(* IEC 61131-3 sources: POMIRTS_lab3/AS/Library_2/MTRegister/V2.00.0, 3 files *)

(* ---- MTRegister.typ ---- *)
TYPE
	MTRegisterControllerInternalType : 	STRUCT  (*Data for internal use.*)
		CycleTime : REAL; (*Task cycle time. Unit: [s].*)
		ImageLength : REAL; (*Data for internal use.*)
		WebLength : REAL; (*Data for internal use.*)
		SensorPosition : REAL; (*Data for internal use.*)
		MaxVelocityCorrection : REAL; (*Data for internal use.*)
		ResponseRate : REAL; (*Data for internal use.*)
		ResponseOvershoot : REAL; (*Data for internal use.*)
		PrefilterOut : REAL; (*Data for internal use.*)
		ControlStateVariable : REAL; (*Data for internal use.*)
		ControllerParameter : ARRAY[0..2]OF REAL; (*Data for internal use.*)
		ActSystemSampleTime : REAL; (*Data for internal use.*)
		UpdateParametersValid : BOOL; (*Data for internal use.*)
		InitParametersValid : BOOL; (*Data for internal use.*)
		ParametersValid : BOOL; (*Data for internal use.*)
		EnableOld : BOOL; (*Data for internal use.*)
		UpdateOld : BOOL; (*Data for internal use.*)
		InitControllerOld : BOOL; (*Data for internal use.*)
		TriggerOld : BOOL; (*Data for internal use.*)
		ResetOld : BOOL; (*Data for internal use.*)
	END_STRUCT;
	MTRegisterControlModeEnum :
		( (*Mode for the longitudinal register error.*)
		mtPRN_KEY_COLOR := 0, (*Key color mode.*)
		mtPRN_SEQUENTIAL_COLOR := 1 (*Sequential color mode.*)
		);
	MTRegisterDecouplingInternalType : 	STRUCT  (*Data for internal use.*)
		CycleTime : REAL; (*Task cycle time. Unit: [s].*)
		ParametersValid : BOOL; (*Data for internal use.*)
		UpdateOld : BOOL; (*Data for internal use.*)
		EnableOld : {REDUND_UNREPLICABLE} BOOL; (*Data for internal use.*)
		Parameters : {REDUND_UNREPLICABLE} MTRegisterSystemType; (*Data for internal use.*)
		Strain : ARRAY[0..19]OF REAL; (*Data for internal use.*)
		DelayedStrain : ARRAY[0..19]OF REAL; (*Data for internal use.*)
		DelayedChangingStrain : ARRAY[0..19]OF REAL; (*Data for internal use.*)
		NumberOfBufferElements : UINT; (*Data for internal use.*)
		UpdateEpsBuffer : ARRAY[0..18]OF BOOL; (*Data for internal use.*)
		UpdateEpsDerBuffer : ARRAY[0..18]OF BOOL; (*Data for internal use.*)
		EpsBuffer : ARRAY[0..18]OF MTRegisterTransDelayBufferType; (*Data for internal use.*)
		EpsDerBuffer : ARRAY[0..18]OF MTRegisterTransDelayBufferType; (*Data for internal use.*)
		TransportDelayDerivation : ARRAY[0..18]OF REAL; (*Data for internal use.*)
	END_STRUCT;
	MTRegisterSimulationModelIntType : 	STRUCT  (*Data for internal use.*)
		CycleTime : REAL; (*Task cycle time. Unit: [s].*)
		ParametersValid : BOOL; (*Data for internal use.*)
		UpdateOld : BOOL; (*Data for internal use.*)
		EnableOld : {REDUND_UNREPLICABLE} BOOL; (*Data for internal use.*)
		Parameters : {REDUND_UNREPLICABLE} MTRegisterSimulationModelType; (*Data for internal use.*)
		Strain : ARRAY[0..19]OF LREAL; (*Data for internal use.*)
		DelayedStrain : ARRAY[0..19]OF LREAL; (*Data for internal use.*)
		KeyError : ARRAY[0..19]OF REAL; (*Data for internal use.*)
		SequentialError : ARRAY[0..19]OF REAL; (*Data for internal use.*)
		MaterialBreak : ARRAY[0..19]OF BOOL; (*Data for internal use.*)
		RestOfMaterial : ARRAY[0..19]OF REAL; (*Data for internal use.*)
		RegisterError : ARRAY[0..19]OF REAL; (*Data for internal use.*)
		DeltaPos : ARRAY[0..19]OF REAL; (*Data for internal use.*)
		Trigger : ARRAY[0..19]OF BOOL; (*Data for internal use.*)
		NumberEpsBufferElements : USINT; (*Data for internal use.*)
		UpdateEpsBuffer : ARRAY[0..18]OF BOOL; (*Data for internal use.*)
		EpsBuffer : ARRAY[0..18]OF MTRegisterTransDelayLRBufferType; (*Data for internal use.*)
	END_STRUCT;
	MTRegisterSimulationModelType : 	STRUCT  (*Parameter for the simulation model.*)
		NumberOfPrintingUnits : USINT; (*Number of printing units.*)
		ImageLength : DINT; (*Circumference of printing cylinders.*)
		WebLength : ARRAY[0..19]OF DINT; (*Web length between PU#i and PU#i-1. Unit: [µm].*)
		SensorPosition : ARRAY[0..19]OF DINT; (*Distance from printing unit to register mark sensor LSi. Unit: [µm].*)
		Mode : ARRAY[0..19]OF MTRegisterControlModeEnum; (*Control mode array.*)
		TensionIn : REAL; (*Feed tension prior to the first printing unit. Unit: [N].*)
		Noise : BOOL; (*Measurement noise is enabled or disabled.*)
	END_STRUCT;
	MTRegisterSystemType : 	STRUCT  (*System parameters for the decoupling.*)
		NumberOfPrintingUnits : USINT; (*Number of printing units. *)
		WebLength : ARRAY[0..19]OF DINT; (*Web length between PU#i und PU#i-1. Unit: [µm].*)
		Mode : ARRAY[0..19]OF MTRegisterControlModeEnum; (*Control mode array.*)
		AccelerationCompensation : BOOL; (*Compensation of additional acceleration terms.*)
	END_STRUCT;
	MTRegisterTransDelayBufferType : 	STRUCT  (*Buffer parameters for the transport delay.*)
		NumberOfBufferElements : UDINT; (*Data for internal use.*)
		CurrentIndex : UDINT; (*Data for internal use.*)
		DelayIndex : UDINT; (*Data for internal use.*)
		DiffIndex : DINT; (*Data for internal use.*)
		Integration : LREAL; (*Data for internal use.*)
		DataIn : REFERENCE TO REAL; (*Data for internal use.*)
		DataTt : REFERENCE TO REAL; (*Data for internal use.*)
		TimeDelay : REAL; (*Data for internal use.*)
		TransportDelay : REAL; (*Data for internal use.*)
		TransportDelayDerivation : REAL; (*Data for internal use.*)
		MaxDelayTime : REAL; (*Data for internal use.*)
	END_STRUCT;
	MTRegisterTransDelayLRBufferType : 	STRUCT  (*Buffer parameters for the transport delay.*)
		NumberOfBufferElements : UDINT; (*Data for internal use.*)
		CurrentIndex : UDINT; (*Data for internal use.*)
		DelayIndex : UDINT; (*Data for internal use.*)
		DiffIndex : DINT; (*Data for internal use.*)
		Integration : LREAL; (*Data for internal use.*)
		DataIn : REFERENCE TO LREAL; (*Data for internal use.*)
		DataTt : REFERENCE TO REAL; (*Data for internal use.*)
		TimeDelay : REAL; (*Data for internal use.*)
		TransportDelay : REAL; (*Data for internal use.*)
		TransportDelayDerivation : REAL; (*Data for internal use.*)
		MaxDelayTime : REAL; (*Data for internal use.*)
	END_STRUCT;
END_TYPE

(* ---- MTRegister.fun ---- *)
{REDUND_OK} FUNCTION_BLOCK MTRegisterController (*PID controller for mark to mark register control in rotogravure printing presses.*)
	VAR_INPUT
		Enable : BOOL; (*The function block is active as long as this input is set.*)
		WebLength : DINT; (*Web length to previous printing unit Lij. Unit: [µm]. *)
		ImageLength : DINT; (*Circumference of printing cylinder. Unit: [µm]. *)
		SensorPosition : DINT; (*Distance from printing unit to register mark sensor LSi. Unit: [µm]. *)
		MaxVelocityCorrection : REAL; (*Positive and negative limit of controller output. Unit: [µm/s]. *)
		Update : BOOL; (*Parameters are updated on a rising edge of the input.*)
		SetLineVelocity : REAL; (*Set line velocity. Unit: [µm/s].*)
		SetRegisterPosition : DINT; (*Set register position. Unit: [µm].*)
		ActRegisterPosition : DINT; (*Actual register position. Unit: [µm].*)
		Trigger : BOOL; (*Every rising edge of "Trigger" a new output "VelocityCorrection" is calculated.*)
		ResponseRate : REAL; (*Defines the time constant of the control loop. *)
		ResponseOvershoot : REAL; (*Defines the tendency to oscillate of the control loop. *)
		InitController : BOOL; (*Initializes the control parameters according to the inputs "ResponseRate" and "ResponseOvershoot" at a positive edge.*)
		Invert : BOOL; (*Inverts the controller output.*)
		Hold : BOOL; (*Freezes the function block.*)
		Reset : BOOL; (*Every rising edge of "Reset" the controller states are reset to zero.*)
	END_VAR
	VAR_OUTPUT
		Active : BOOL; (*The function block is active.*)
		Error : BOOL; (*Error occurred during operation.*)
		StatusID : DINT; (*Status information.*)
		UpdateDone : BOOL; (*Parameters updated.*)
		VelocityCorrection : REAL; (*Actual correction velocity. Unit: [µm/s].*)
		InitDone : BOOL; (*Controller parameters initialized successfully.*)
	END_VAR
	VAR
		Internal : MTRegisterControllerInternalType; (*Data for internal use.*)
	END_VAR
END_FUNCTION_BLOCK

{REDUND_CONTEXT} FUNCTION_BLOCK MTRegisterDecoupling (*Decoupling network for velocities of printing cylinders in rotogravure printing presses.*)
	VAR_INPUT
		Enable : BOOL; (*The function block is active as long as this input is set.*)
		Parameters : MTRegisterSystemType; (*System parameters.*)
		Update : BOOL; (*Parameters are updated on a rising edge of the input.*)
		VelocityCorrectionIn : ARRAY[0..19] OF REAL; (*Correction velocity input. Unit: [µm/s].*)
		SetLineVelocity : REAL; (*Set line velocity. Unit: [µm/s].*)
	END_VAR
	VAR_OUTPUT
		Active : BOOL; (*The function block is active.*)
		Error : BOOL; (*Error occurred during operation.*)
		StatusID : DINT; (*Status information.*)
		UpdateDone : BOOL; (*Parameters updated.*)
		VelocityCorrectionOut : ARRAY[0..19] OF REAL; (*Decoupled correction velocity. Unit: [µm/s].*)
	END_VAR
	VAR
		Internal : MTRegisterDecouplingInternalType; (*Data for internal use.*)
	END_VAR
END_FUNCTION_BLOCK

{REDUND_CONTEXT} FUNCTION_BLOCK MTRegisterSimulationModel (*Simulation model of a rotogravure printing press.*)
	VAR_INPUT
		Enable : BOOL; (*The function block is active as long as this input is set.*)
		Parameters : MTRegisterSimulationModelType; (*Parameters for the simulation model.*)
		Update : BOOL; (*Parameters are updated on a rising edge of the input.*)
		SetLineVelocity : REAL; (*Set line velocity. Unit: [µm/s].*)
		ActVelocity : ARRAY[0..19] OF REAL; (*Actual velocity of the printing cylinder. Unit: [µm/s].*)
	END_VAR
	VAR_OUTPUT
		Active : BOOL; (*The function block is active.*)
		Error : BOOL; (*Error occurred during operation.*)
		StatusID : DINT; (*Status information.*)
		UpdateDone : BOOL; (*Parameters updated.*)
		ActRegisterPosition : ARRAY[0..19] OF DINT; (*Actual register position. Unit: [µm].*)
		Trigger : ARRAY[0..19] OF BOOL; (*Rising edge indicates new "ActRegisterPosition" value.*)
		MaterialBreak : BOOL; (*Material breakage has been detected.*)
	END_VAR
	VAR
		Internal : MTRegisterSimulationModelIntType; (*Data for internal use.*)
	END_VAR
END_FUNCTION_BLOCK

(* ---- MTRegister.var ---- *)
(*Error: MTRegister*)
VAR CONSTANT
	mtPRN_ERR_WEB_LENGTH_INVALID : DINT := -1058006164; (*The selected web length is invalid.*)
END_VAR
(*Error: MTRegisterSimulationModel and MTRegisterDecoupling*)
VAR CONSTANT
	mtPRN_ERR_NR_OF_PRINTING_UNITS : DINT := -1058006144; (*The selected number of printing units is invalid.*)
	mtPRN_ERR_REGISTER_MODE_INVALID : DINT := -1058006138; (*The selected mode is invalid.*)
END_VAR
(*Error: MTRegisterSimulationModel*)
VAR CONSTANT
	mtPRN_ERR_TENSION_IN_INVALID : DINT := -1058006143; (*The input tension before the first printing unit is invalid.*)
	mtPRN_ERR_MATERIAL_BREAK : DINT := -1058006137; (*Material failure was detected.*)
END_VAR
(*Error: MTRegisterSimulationModel and MTRegisterController*)
VAR CONSTANT
	mtPRN_ERR_IMAGE_LENGTH_INVALID : DINT := -1058006142; (*The circumference of the printing cylinder is invalid.*)
	mtPRN_ERR_SENSOR_POSITION : DINT := -1058006141; (*The selected distance between the printing unit and the register mark sensor is invalid.*)
END_VAR
(*Error: MTRegisterController*)
VAR CONSTANT
	mtPRN_ERR_RESPONSE_RATE_INVALID : DINT := -1058006162; (*The selected value for the parameter that defines the time constant of the control loop is invalid.*)
	mtPRN_ERR_MAX_VEL_CORRECTION : DINT := -1058006140; (*The selected output limit for the correction velocity is invalid.*)
	mtPRN_ERR_RESPONSE_OVERSHOOT : DINT := -1058006139; (*The selected value for the parameter that defines the tendency of the control loop to overshoot is invalid.*)
END_VAR
(*Warning: MTRegister*)
VAR CONSTANT
	mtPRN_WRN_WEB_LENGTH_INVALID : DINT := -2131747988; (*The selected web length is invalid.*)
END_VAR
(*Warning: MTRegisterSimulationModel and MTRegisterDecoupling*)
VAR CONSTANT
	mtPRN_WRN_NR_OF_PRINTING_UNITS : DINT := -2131747968; (*The selected number of printing units is invalid.*)
	mtPRN_WRN_REGISTER_MODE_INVALID : DINT := -2131747962; (*The selected mode is invalid.*)
END_VAR
(*Warning: MTRegisterSimulationModel*)
VAR CONSTANT
	mtPRN_WRN_TENSION_IN_INVALID : DINT := -2131747967; (*The input tension before the first printing unit is invalid.*)
END_VAR
(*Warning: MTRegisterSimulationModel and MTRegisterController*)
VAR CONSTANT
	mtPRN_WRN_IMAGE_LENGTH_INVALID : DINT := -2131747966; (*The circumference of the printing cylinder is invalid.*)
	mtPRN_WRN_SENSOR_POSITION : DINT := -2131747965; (*The selected distance between the printing unit and the register mark sensor is invalid.*)
END_VAR
(*Warning: MTRegisterController*)
VAR CONSTANT
	mtPRN_WRN_RESPONSE_RATE_INVALID : DINT := -2131747986; (*The selected value for the parameter that defines the time constant of the control loop is invalid.*)
	mtPRN_WRN_CTRL_PAR_CALCULATION : DINT := -2131747982; (*Calculation of the control parameters has failed.*)
	mtPRN_WRN_MAX_VEL_CORRECTION : DINT := -2131747964; (*The selected output limit for the correction velocity is invalid.*)
	mtPRN_WRN_RESPONSE_OVERSHOOT : DINT := -2131747963; (*The selected value for the parameter that defines the tendency of the control loop to overshoot is invalid.*)
END_VAR
